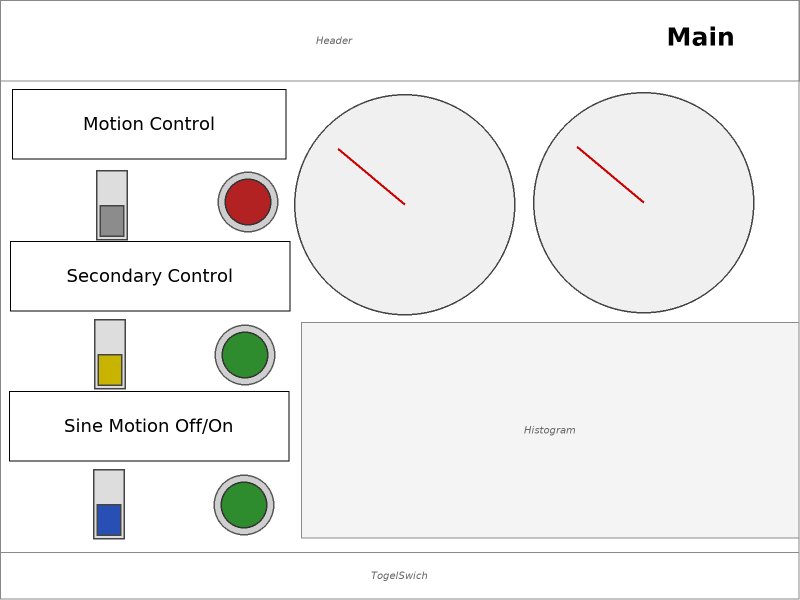
VISUALIZATION Main_screen  // 800x600
    Frame (-132,0 932x81)
        shows Header()
    Histogram (301,322 498x216), scale format: %.1f, scale 0..2
        p1518820177: G_Sensors.fPayLoadPosition
        p102497268: G_Sensors.fPayLoadPosition
    Meter360 (294,93 221x223), value: G_Sensors.fPressureWinchA, style: Meter-Meter360-Gray, scale format: %.1f, scale 0..100
        p518627256: PA bar
    Meter360 (533,91 221x223), value: G_Sensors.fPressureWinchB, style: Meter-Meter360-Gray, scale format: %.1f, scale 0..100
        p518627256: PB bar
    Frame (0,552 799x47)
        shows TogelSwich()
    Textfield (623,20 156x33), "Main"
    DipSwitch (30,319 160x70), variable: HMI.bActvateSMC, behaviour: TOGGLE, style: Switch-DipSwitch-Yellow
    Rectangle (10,241 280x70), "Secondary Control"
    Lamp1 (210,320 70x70), variable: not HMI.bActvateSMC, style: Lamp-Lamp1-Red
    Lamp1 (210,320 70x70), variable: HMI.bActvateSMC, invisible if: not HMI.bActvateSMC, style: Lamp-Lamp1-Green
    DipSwitch (29,469 160x70), variable: HMI.bSwicher, behaviour: TOGGLE, style: Switch-DipSwitch-Blue
    Rectangle (9,391 280x70), "Sine Motion Off/On"
    Lamp1 (209,470 70x70), variable: not HMI.bSwicher, style: Lamp-Lamp1-Red
    Lamp1 (209,470 70x70), variable: HMI.bSwicher, invisible if: not HMI.bSwicher, style: Lamp-Lamp1-Green
    Lamp1 (213,167 70x70), variable: HMI.bStartTB, invisible if: not HMI.bStartTB, style: Lamp-Lamp1-Green
    DipSwitch (32,170 160x70), variable: HMI.bStartTB, behaviour: TOGGLE, style: Switch-DipSwitch-Gray
    Rectangle (12,89 274x70), "Motion Control"
    Lamp1 (213,167 70x70), variable: not HMI.bStartTB, invisible if: HMI.bStartTB, style: Lamp-Lamp1-Red
END_VISUALIZATION

(* stored: Version 1.1.0.1, ProductVersion 3.1.4024.12
   Visu Main_screen: Id {9b1380ab-3734-4573-ab0a-e510f86d8ad1} *)
